(* CoDeSys 2.3 export: CALLBACKTASKCODENC.EXP *)

(* POU NetVar POUs/CallbackTaskCodeNC, ST *)
FUNCTION CallbackTaskCodeNC : BYTE
VAR_INPUT
	dwEvent			: DWORD;
	dwFilter		: DWORD;
	dwOwner			: DWORD;
END_VAR
(* @TEXT_IMPLEMENTATION := 'ST' *)
g_bCPUStopNetVar := TRUE;
NetVarManager_Udp();
g_bCPUStopNetVar := FALSE;
END_FUNCTION
